FUNCTION_BLOCK FutureSleepCreator IMPLEMENTS I_TaskCreator
VAR_INPUT
END_VAR
VAR_OUTPUT
END_VAR
VAR
	_sleep_time: TIME;
	_p_future : POINTER TO FutureSleep;
END_VAR

{warning 'add method implementation '}
METHOD create_future : I_Future
VAR_INPUT
	(* Specify future name*)
	future_name	: STRING;
END_VAR
_p_future := __NEW(FutureSleep);
_p_future^.future_name := future_name;
_p_future^.sleep_time := _sleep_time;
create_future := _p_future^;
END_METHOD

{warning 'add method implementation '}
METHOD destroy_future : I_Future
VAR_INPUT
	(* Specify future instance whtat you want to delete.*)
	future	: I_Future;
END_VAR
VAR
	_p_future : POINTER TO FutureSleep;
END_VAR
IF __QUERYPOINTER(future, _p_future) THEN
	__DELETE(_p_future);
	IF _p_future = 0  THEN
		destroy_future := 0;
	END_IF
END_IF
END_METHOD

PROPERTY sleep_time : TIME
GET
sleep_time := _p_future^.sleep_time;
END_GET
SET
_sleep_time := sleep_time;
END_SET
END_PROPERTY

END_FUNCTION_BLOCK

(* stored: Version 1.1.0.1, ProductVersion 3.1.4026.17
   POU FutureSleepCreator: Id {e51ff537-6a6c-441a-9c50-d053b3ef0e7c}, SpecialFunc None
   Method create_future: Id {68dc0f33-3150-469d-afb6-499fce7ee32e}
   Method destroy_future: Id {19ea5f74-a9a0-47e9-8242-8d8c60f039bb}
   Property sleep_time: Id {3b9f8465-bfc4-48b1-b1f6-04a38356af9e}
   Get Get: Id {7c4f2e26-1b81-47c4-9ae9-abf10506c853}
   Set Set: Id {5915549c-f74d-45fa-9f29-3ca00808afbd} *)
